Fanuc KAREL source: IO0209.KL

PROGRAM IO0209
%STACKSIZE=65535
%PRIORITY=65535
%NOLOCKGROUP
ROUTINE RTEST FROM IO0209
ROUTINE RTEST
VAR
L1 : ARRAY[3] OF INTEGER
L2 : XYZWPR
L3 : JOINTPOS9
L4 : POSITION
U2C_37 : BOOLEAN -- ASSUMED 2C source type; see uncertainty report
S1 : INTEGER
U2C_39 : REAL -- ASSUMED 2C source type; see uncertainty report
U2C_40 : BOOLEAN -- ASSUMED 2C source type; see uncertainty report
S2 : REAL
BEGIN
U2C_37=TRUE
L1[1]=2
U2C_40=TRUE
S2=1.0
SET_REAL_REG(1,S2,S1)
END RTEST
BEGIN
RTEST
END IO0209
